{attribute 'qualified_only'}
{attribute 'strict'}
{attribute 'to_string'}
TYPE eSequenceState  :
(
	BEREIT	 		:= 0,				// Der Skill ist bereit einen Prozess auszuführen (Startzustand)
	LAUFEND 		:= 1				// Der Skill führt einen Prozess aus
);
END_TYPE

(* stored: Version 1.1.0.1
   DUT eSequenceState: Id {936565d6-d3db-4758-807a-44491b3159a0} *)
